FUNCTION_BLOCK PUBLIC EnumerableInterface_TestSuite EXTENDS TcUnit.FB_TestSuite
VAR
END_VAR

CompileCheckWithMockEnumerable();

METHOD PUBLIC CompileCheckWithMockEnumerable
VAR
	mockEnumerable : MockEnumerable;
	forwardEnumerator : I_ForwardEnumerator;
	isValidResult : BOOL;
END_VAR
TEST('CompileCheckWithMockEnumerable');

forwardEnumerator := mockEnumerable.GetEnumerator();
isValidResult := forwardEnumerator.IsValid;
forwardEnumerator.Dispose();

AssertFalse(
	Condition := isValidResult,
	Message := 'IsValid did not match the mock set value'
);

TEST_FINISHED();
END_METHOD

END_FUNCTION_BLOCK

(* stored: Version 1.1.0.1, ProductVersion 3.1.4024.12
   POU EnumerableInterface_TestSuite: Id {9c41e908-1d0b-4310-8742-53a2d0bb79f0}, SpecialFunc None
   Method CompileCheckWithMockEnumerable: Id {b31b1045-76da-442d-a56e-cc3cb80cf92f} *)
